// TwinCAT 3 PLC project Functions
// ProgramVersion: 3.1.4023.0
// libraries:
//   Tc2_Standard, * (Beckhoff Automation GmbH)
//   Tc2_System, * (Beckhoff Automation GmbH)
//   Tc3_Module, * (Beckhoff Automation GmbH)
// project tree:
//   / PlcTask.TcTTO
//   POUs/ Celsius_To_Fahrenheit.TcPOU, Greater_Smaller.TcPOU, MAIN.TcPOU, MAIN_Greater_Smaller.TcPOU, SwapNums.TcPOU
// (motion and I/O tree: see PLC project arrays1)
// real-time tasks:
//   TASK PlcTask: cycle T#10ms, priority 20, ADS port 350
//   TASK PlcTask1: cycle T#10ms, priority 21, ADS port 351
//   TASK PlcTask2: cycle T#10ms, priority 22, ADS port 352
//   TASK PlcTask3: cycle T#10ms, priority 23, ADS port 353

CONFIGURATION Functions
    RESOURCE PLC ON TwinCAT3
        TASK PlcTask(INTERVAL := T#10ms, PRIORITY := 22);
        PROGRAM MAIN WITH PlcTask : MAIN;
    END_RESOURCE
END_CONFIGURATION

// ---- POUs/MAIN.TcPOU
PROGRAM MAIN
VAR
	fFahrenheit : REAL;
END_VAR

fFahrenheit := Celsius_To_Fahrenheit(fCelsius := 5.0);

END_PROGRAM

// ---- POUs/Celsius_To_Fahrenheit.TcPOU
FUNCTION Celsius_To_Fahrenheit : REAL
VAR_INPUT
	fCelsius : REAL;
END_VAR
VAR
// scratch pad where program variables are stored.
END_VAR

Celsius_To_Fahrenheit := fCelsius * 1.8 + 32.0;

END_FUNCTION

// ---- POUs/Greater_Smaller.TcPOU
FUNCTION Greater_Smaller
VAR_INPUT
	nNumber1 : INT;
	nNumber2 : INT;
END_VAR
VAR_OUTPUT
	nGreater : INT;
	nSmaller : INT;
END_VAR

IF nNumber1 > nNumber2 THEN
	nGreater := nNumber1;
	nSmaller := nNumber2;
ELSE
	nGreater := nNumber2;
	nSmaller := nNumber1;
END_IF

END_FUNCTION

// ---- POUs/MAIN_Greater_Smaller.TcPOU
PROGRAM MAIN_Greater_Smaller
VAR
	nReturnGreater : INT;
	nReturnSmaller : INT;
	
	nA : INT := 5;
	nB : int := 15;
END_VAR

(*Note how to assign output values from function to variables using '=>'*)
Greater_Smaller(nNumber1 := 8, nNumber2 := 15, nGreater => nReturnGreater, nSmaller => nReturnSmaller);

SwapNums(nNumber1 := nA, nNumber2 := nB);

END_PROGRAM

// ---- POUs/SwapNums.TcPOU
FUNCTION SwapNums
VAR_IN_OUT
	nNumber1 : INT;
	nNumber2 : INT;
END_VAR
VAR
	nNumberTemp : INT;
END_VAR

nNumberTemp := nNumber1;
nNumber1 := nNumber2;
nNumber2 := nNumberTemp;

END_FUNCTION
